{attribute 'pack_mode' := '1'}
TYPE TOperatorReq :
STRUCT
	abFreeLoaderLift			: ARRAY[0..1] OF BOOL;
	bSampleRequest			: BOOL;
END_STRUCT
END_TYPE

(* stored: Version 1.1.0.1, ProductVersion 3.1.4022.12
   DUT TOperatorReq: Id {9f7a121e-82d1-4b06-bb1d-574087243055} *)
